(* CoDeSys 2.3 export: CLIENT_REPLY.EXP *)

(* Data type *)
TYPE CLIENT_REPLY :
STRUCT
	diBytesReceived			: DINT;
	dwIPAddress				: DWORD;
	stIPAddressTransmitter	: STRING(20);
END_STRUCT
END_TYPE
